// TIA Portal V20 export
TYPE "LER_typeHotPressTrackingData"
// stored: Access Published
   STRUCT
      finished { ExternalWritable := 'False'} : Bool;
      result { ExternalWritable := 'False'} : Bool;
   END_STRUCT;
END_TYPE
